// TIA Portal V19 export
VAR_GLOBAL   // PLC tag table "TT - Transport"
   iTransportSenDown_h1 AT %I1.4 : Bool;
   iTransportSenUp_h0 AT %I1.5 : Bool;
   iTransportSenAtPlate_i0 AT %I2.2 : Bool;
   iTransportSenAtCart_i1 AT %I2.3 : Bool;
   "oTransportVenCilDown_A+" AT %Q1.2 : Bool;
   "oTransportVenCilCart_I+" AT %Q1.3 : Bool;
   "oTransportVenGripClosed_J+" AT %Q1.4 : Bool;
END_VAR
